FUNCTION_BLOCK E_TMIN (* Forwards Events with a minimum inter-arrival time between EI events *)
  (* Standard: 61499-2; Description: Copyright (c) 2026 HR Agrartechnik GmbH This program and the accompanying materials are made available under the terms of the Eclipse Public License 2.0 which is available at https://www.eclipse.org/legal/epl-2.0/ SPDX-License-Identifier: EPL-2.0 *)
  (* Version 1.0, 2026-05-14, Franz Höpfinger, HR Agrartechnik GmbH, Initial API *)
  PACKAGE iec61499::events;
  IMPORT eclipse4diac::core::TypeHash;
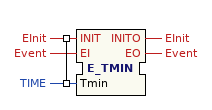
  EVENT_INPUT
    INIT : EInit WITH Tmin; (* Initialization Request *)
    EI;
  END_EVENT
  EVENT_OUTPUT
    INITO : EInit; (* Initialization Confirm *)
    EO;
  END_EVENT
  VAR_INPUT
    Tmin : TIME; (* Minimum inter-arrival time between EI events *)
  END_VAR
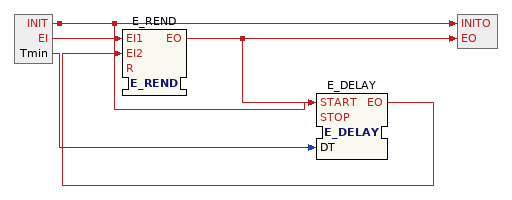
  FBS
    E_REND : iec61499::events::E_REND;
    E_DELAY : iec61499::events::E_DELAY;
  END_FBS
  EVENT_CONNECTIONS
    E_DELAY.EO TO E_REND.EI2;
    E_REND.EO TO E_DELAY.START;
    INIT TO INITO;
    INIT TO E_DELAY.START;
    EI TO E_REND.EI1;
    E_REND.EO TO EO;
  END_CONNECTIONS
  DATA_CONNECTIONS
    Tmin TO E_DELAY.DT;
  END_CONNECTIONS
END_FUNCTION_BLOCK
